Universal Robots URScript: Project1pick.script

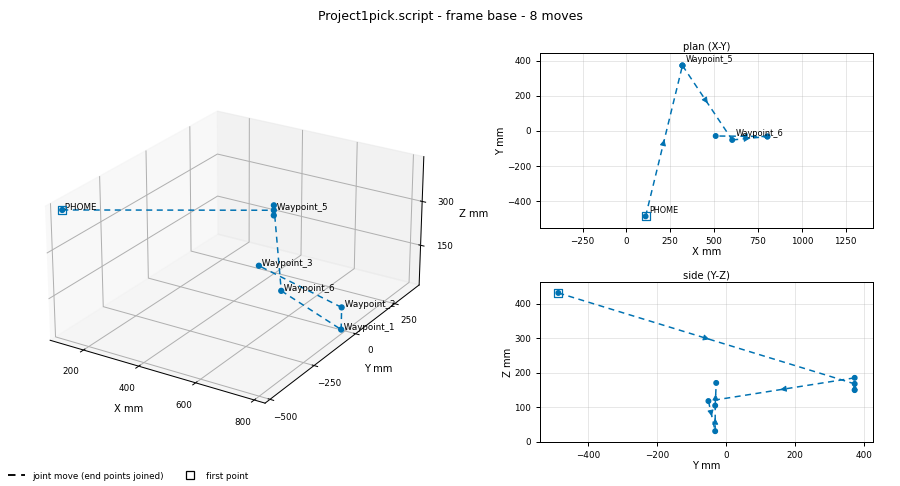
[picture p0: tool path of Project1pick.script in frame base, 8 of 8 moves have a stored position in this frame; points joined in program order, loops and branches not executed]
def Project1pick():
  set_safety_mode_transition_hardness(0)
  modbus_add_signal("127.0.0.1", 255, 1, 2, "MODBUS_1", False)
  modbus_set_signal_update_frequency("MODBUS_1", 10)
  modbus_add_signal("127.0.0.1", 255, 128, 0, "atLocation", False)
  modbus_set_signal_update_frequency("atLocation", 10)
  modbus_add_signal("10.241.34.56", 1, 1009, 3, "MODBUS_2", False)
  modbus_set_signal_update_frequency("MODBUS_2", 10)
  modbus_set_runstate_dependent_choice("MODBUS_2",0)
  set_standard_analog_input_domain(0, 1)
  set_standard_analog_input_domain(1, 1)
  set_tool_analog_input_domain(0, 0)
  set_tool_analog_input_domain(1, 0)
  set_analog_outputdomain(0, 0)
  set_analog_outputdomain(1, 0)
  set_input_actions_to_default()
  set_tcp(p[0.0,0.0,0.0,0.0,0.0,0.0])
  set_payload(1.0)
  set_gravity([0.0, 0.0, 9.82])
  step_count_39999969_9eca_48ce_a050_47ed1e067633 = 0.0
  thread Step_Counter_Thread_00328349_14f1_4d2f_a40a_433a0710b75e():
    while (True):
      step_count_39999969_9eca_48ce_a050_47ed1e067633 = step_count_39999969_9eca_48ce_a050_47ed1e067633 + 1.0
      sync()
    end
  end
  run Step_Counter_Thread_00328349_14f1_4d2f_a40a_433a0710b75e()
  set_tool_voltage(0)
  $ 1 "Robot Program"
  $ 2 "Set DO[0]=Off"
  set_standard_digital_out(0, False)
  $ 3 "MoveJ"
  $ 4 "PHOME" "breakAfter"
  movej(get_inverse_kin(p[.109126988750, -.486919972196, .431878117393, .000159938141, 3.141482481273, -.000243878919], qnear=[1.570730447769165, -1.570796314870016, 1.5707850456237793, -1.5709403196917933, -1.570686165486471, 3.5952674807049334E-5]), a=1.3962634015954636, v=1.0471975511965976)
  $ 5 "Waypoint_5" "breakAfter"
  movej(get_inverse_kin(p[.319215129822, .373245107778, .168002937454, .034421956458, 3.130169751828, .057990472087], qnear=[-2.506416622792379, -1.367345158253805, 2.0854063034057617, -2.319710079823629, -1.547663990651266, -4.054863278065817]), a=1.3962634015954636, v=1.0471975511965976)
  $ 6 "Waypoint_7" "breakAfter"
  movej(get_inverse_kin(p[.319229208460, .373190364173, .149809568861, .034571477834, 3.130150061837, .057984580479], qnear=[-2.506524149571554, -1.333916966115133, 2.1042871475219727, -2.3720300833331507, -1.547675911580221, -4.054875198994772]), a=1.3962634015954636, v=1.0471975511965976)
  $ 7 "Wait: 0.5"
  sleep(0.5)
  $ 8 "Set DO[0]=On"
  set_standard_digital_out(0, True)
  $ 9 "Wait: 0.5"
  sleep(0.5)
  $ 10 "lift" "breakAfter"
  movej(get_inverse_kin(p[.319243664558, .373173483176, .185478439030, .034587227000, 3.129983312472, .058056954711], qnear=[-2.5065601507769983, -1.397433106099264, 2.065566062927246, -2.2699530760394495, -1.5477359930621546, -4.054899040852682]), a=1.3962634015954636, v=1.0471975511965976)
  $ 11 "Waypoint_6" "breakAfter"
  movej(get_inverse_kin(p[.602971949846, -.051245048280, .118113577118, -2.185325154958, -2.244004470980, -.001678195271], qnear=[-3.4084914366351526, -1.0625837484942835, 1.7848587036132812, -2.2854445616351526, -1.5653532187091272, -3.4350064436541956]), a=1.3962634015954636, v=1.0471975511965976)
  $ 12 "Waypoint_1" "breakAfter"
  movej(get_inverse_kin(p[.803631980481, -.031647524643, .030647552201, -2.197009595446, -2.240727017917, -.005130119599], qnear=[-3.317570511494772, -0.546734635029928, 1.0731253623962402, -2.096156899129049, -1.566131893788473, -3.3372748533831995]), a=1.3962634015954636, v=1.0471975511965976)
  $ 13 "Wait: 0.5"
  sleep(0.5)
  $ 14 "Set DO[0]=Off"
  set_standard_digital_out(0, False)
  $ 15 "Wait: 0.5"
  sleep(0.5)
  $ 16 "Waypoint_2" "breakAfter"
  movej(get_inverse_kin(p[.803650718001, -.031602234131, .104989727519, -2.197030859726, -2.240856793207, -.005245787943], qnear=[-3.317510430012838, -0.6368988196002405, 1.0418457984924316, -1.9748438040362757, -1.566131893788473, -3.3372626940356653]), a=1.3962634015954636, v=1.0471975511965976)
  $ 17 "Waypoint_3" "breakAfter"
  movej(get_inverse_kin(p[.508862438714, -.028636304084, .170727470542, -2.196986498727, -2.240712990886, -.005196109745], qnear=[-3.414398733769552, -1.332874600087301, 2.0206899642944336, -2.2571328322040003, -1.5662038961993616, -3.43410832086672]), a=1.3962634015954636, v=1.0471975511965976)
end
